INTERFACE I_WriteParameter EXTENDS I_Status

METHOD WriteParameter
VAR_INPUT
    ParameterNumber : MC_AxisParameter;
    ParameterValue	: LREAL;
END_VAR
END_METHOD

END_INTERFACE

(* stored: Version 1.1.0.1
   Itf I_WriteParameter: Id {e84a3142-abbc-454b-a28f-e59f4606fe82}
   Method WriteParameter: Id {56820ef8-d494-4985-91bc-3e70e63092e8} *)
